{attribute 'GeneratedUsingTerminal: EL3102-0000-0016'}
{attribute addProperty BoxType "EL3102-0000-0016"}
{attribute addProperty Id "AI_Standard_Channel_1AT %I*AI_Standard_Channel_A8DF64E310AI_Standard_Channel_2AT %I*AI_Standard_Channel_A8DF64E310WcStateAT %I*WcState_9091E0EB2InfoDataAT %I*InfoData_94A18F5E2"}
{attribute addProperty CRC "4240555915"}
{attribute addProperty Size "24"}
TYPE EL3102_FCC1BF8B EXTENDS EtcSlaveTerminalBase_947E5A46 :
STRUCT
	{attribute addProperty Name "AI_Standard_Channel_1"}
	AI_Standard_Channel_1 : AI_Standard_Channel_A8DF64E3;
	{attribute addProperty Name "AI_Standard_Channel_2"}
	AI_Standard_Channel_2 : AI_Standard_Channel_A8DF64E3;
	{attribute addProperty Name "WcState"}
	WcState : WcState_9091E0EB;
	{attribute addProperty Name "InfoData"}
	InfoData : InfoData_94A18F5E;
END_STRUCT
END_TYPE

(* stored: Version 1.2.0.0, ProductVersion 3.1.4024.9
   DUT EL3102_FCC1BF8B: Id {9c1aa927-2a86-4f1e-a51a-8130d0390eaa} *)
